// TwinCAT 3 PLC project Ampelschaltung
// libraries:
//   Tc2_Standard, * (Beckhoff Automation GmbH)
//   Tc2_Standard, * (Beckhoff Automation GmbH)
//   Tc2_System, * (Beckhoff Automation GmbH)
//   Tc2_System, * (Beckhoff Automation GmbH)
//   Tc3_Module, * (Beckhoff Automation GmbH)
//   Tc3_Module, * (Beckhoff Automation GmbH)
// project tree:
//   Global Variables/ Global_Variables.TcGVL, Variable_Configuration.TcGVL
//   / GlobalImagePool.TcGIPO (not stored), GlobalTextList.TcGTLO, Standard.TcTTO, Visualisierungsmanager.TcVMO (not stored)
//   POUs/ fb_Blink.TcPOU, MAIN.TcPOU
//   Visualizations/ Ende.TcVIS, Kreuzung.TcVIS

CONFIGURATION Ampelschaltung
    RESOURCE PLC ON TwinCAT3
        TASK Standard(INTERVAL := T#10ms, PRIORITY := 20);
        PROGRAM MAIN WITH Standard : MAIN;
    END_RESOURCE
END_CONFIGURATION

// ---- Global Variables/Global_Variables.TcGVL
{attribute 'Tc2GvlVarNames'}
VAR_GLOBAL
END_VAR

// ---- Global Variables/Variable_Configuration.TcGVL
{attribute 'Tc2GvlVarNames'}
VAR_CONFIG
END_VAR

// ---- POUs/MAIN.TcPOU
PROGRAM MAIN
VAR

	bON : BOOL;
	diStep : INT;
	bEndeInvisible : BOOL := TRUE;
	bOK : BOOL := FALSE;
	iPhase : REAL;
	bNacht : BOOL;

	(*Ampel Nord-Süd*)
	bNS_rot : BOOL;
	bNS_orange : BOOL;
	bNS_gruen : BOOL;

	(*Ampel West-Ost*)
	bWO_rot : BOOL;
	bWO_orange : BOOL;
	bWO_gruen : BOOL;

	(*Fussgängerampeln Nord-Süd*)
	bFGNS_rot : BOOL;
	bFGNS_gruen : BOOL;
	bFG : BOOL;

	(*Timer*)
	t1 : TON;

	t3 : TON;
	t2 : TON;

END_VAR

t1();

t3.IN := (t2.Q = FALSE);
t2.IN := t3.Q;

t3(PT:=T#3S);
t2(PT:=t#1s);


IF bON = TRUE AND diStep = 0
THEN
	diStep := 1000;

ELSIF bOn = FALSE
THEN
	diStep := 0;
END_IF


CASE diStep OF

0:
(*Idle*)
	bNS_rot:=FALSE;
	bNS_orange := FALSE;
	bNS_gruen := FALSE;

	bWO_rot:=FALSE;
	bWO_orange:=FALSE;
	bWO_gruen:=FALSE;
	bOK:=FALSE;
	bEndeInvisible := TRUE;

	bfgns_gruen := FALSE;
	bfgns_rot:= FALSE;

	t1.IN := FALSE;

	iPhase := 0;




1000:
(*Grünphase Nord-Süd, Rotphase West-Ost*)
	bNS_rot:=FALSE;
	bNS_orange := FALSE;
	bNS_gruen := TRUE;

	bWO_rot:=TRUE;
	bWO_orange:=FALSE;
	bWO_gruen:=FALSE;
	iPhase := 1;
	bfgns_rot := TRUE;

	t1.IN := TRUE;
	t1.PT := T#10000ms;

	IF bFG = TRUE
	THEN
		bfgns_gruen := TRUE;
		bfgns_rot:= FALSE;
	END_IF;

	IF bNacht = TRUE
	THEN
		diStep:=6000;
	END_IF

	IF t1.Q AND bnacht = TRUE
	THEN
		diStep := 6000;
	ELSIF t1.Q AND bNacht = FALSE
	THEN
		t1.IN := FALSE;
		bfgns_gruen := FALSE;
		bfgns_rot := TRUE;
		bFG := FALSE;
		diStep:= 2000;
	END_IF;


2000:
(*Orangephase Nord-Süd*)

	bNS_rot := FALSE;
	bNS_orange := TRUE;
	bNS_gruen := FALSE;

	bWo_rot :=TRUE;
	bWO_orange := TRUE;
	bWO_gruen :=FALSE;

	bFGNS_rot := TRUE;
	bFGNS_gruen := FALSE;

	iPhase := 2;

	t1(IN := bNS_orange, PT := T#5000ms);

		IF t1.Q
		THEN
			t1.IN := FALSE;
			diStep:= 3000;
	END_IF;


3000:
(*Rotphase Nord-Sued, Grünphase West-Ost*)

	bNS_rot:=TRUE;
	bNS_orange := FALSE;
	bNS_gruen := FALSE;

	bWO_rot:=FALSE;
	bWO_orange:=FALSE;
	bWO_gruen:=TRUE;
	iPhase := 3;
	bFGNS_rot := TRUE;

	t1(IN := bNS_rot, PT := T#5000ms);

	IF t1.Q
	THEN
		t1.IN := FALSE;
		diStep:= 4000;
	END_IF;

4000:
(*Rot-Orange-Phase Nord-Sued*)

	bNS_rot:=TRUE;
	bNS_orange := TRUE;
	bNS_gruen := FALSE;

	bWO_rot:=FALSE;
	bWO_orange:=TRUE;
	bWO_gruen:=FALSE;
	bFGNS_rot := TRUE;
	iPhase := 4;

	t1(IN := bNS_rot, PT := T#5000ms);

	IF t1.Q
	THEN
		t1.IN := FALSE;
		diStep:= 1000;
	END_IF;

6000:
(*Nachtmodus*)

	bNS_rot:=FALSE;
	bNS_orange := t3.Q;
	bNS_gruen := FALSE;
	
	bWO_rot:=FALSE;
	bWO_orange:= t3.Q;
	bWO_gruen:=FALSE;

	bFGNS_rot :=FALSE;
	bFGNS_gruen := FALSE;

	IF bNacht = FALSE
	THEN
		t1.IN := FALSE;
		diStep:= 1000;
	END_IF

(*5000:
(*Fenster Ende*)
	bEndeInvisible := FALSE;
	IF bOK
	THEN
		bEndeInvisible := TRUE;
		bON := FALSE;
		diStep := 0;
	END_IF;*)

END_CASE;

END_PROGRAM

// ---- POUs/fb_Blink.TcPOU
FUNCTION_BLOCK fb_Blink
VAR_INPUT
END_VAR
VAR_OUTPUT
END_VAR
VAR
		t1 : TON;
		t2 : TON;
END_VAR




t1.IN := (t2.Q = FALSE);

t2.IN := t1.Q;


t1(PT:=t#1s);
t2(PT:=t#2s); (*FEATUARE*) (*TEST*)

END_FUNCTION_BLOCK

// ---- GlobalTextList.TcGTLO
TEXTLIST GlobalTextList
  225 = 'Bitte drücken'
  117 = 'ENDE'
  226 = 'Nachtmodus'
  118 = 'OK'
  866 = 'ON'
END_TEXTLIST

// ---- Visualizations/Ende.TcVIS
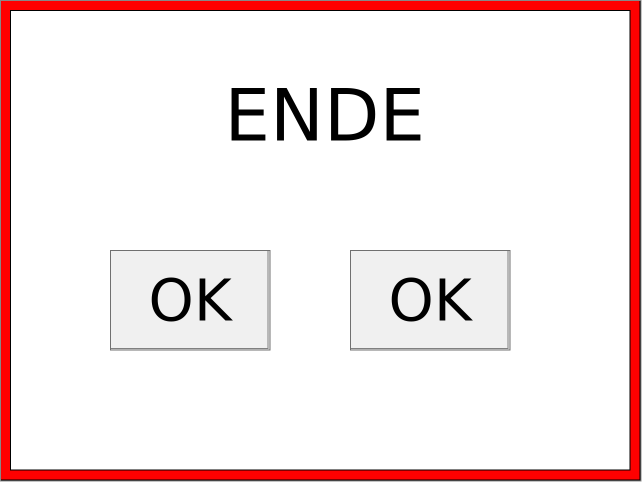
VISUALIZATION Ende  // 642x482
    Rectangle (0,0 640x480)
    Rectangle (10,10 620x460)
    Rectangle (130,50 390x130), "ENDE"
    Button (110,250 160x100), "OK"
        tap MAIN.bOK p1329445385=TRUE
    Button (350,250 160x100), "OK"
        tap MAIN.bOK p1329445385=TRUE
END_VISUALIZATION

// ---- Visualizations/Kreuzung.TcVIS
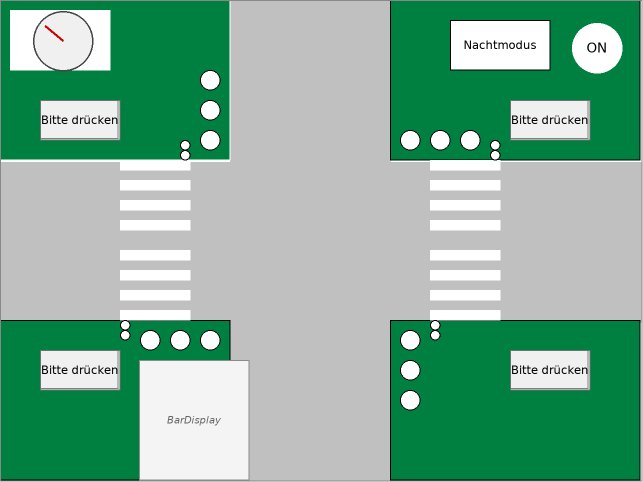
VISUALIZATION Kreuzung  // 643x482
    Rectangle (230,0 160x480)
    Rectangle (1,162 640x160)
    Rectangle (0,0 230x160)
    Rectangle (390,0 250x160)
        tap MAIN.bON
    Rectangle (390,320 250x160)
    Rectangle (0,320 230x160)
    Polyline (230,0)
    Polyline (630,160)
    Polyline (230,480)
    Polyline (630,320)
    Ellipse (200,330 20x20), colour toggle: MAIN.bWO_rot
    Ellipse (170,330 20x20), colour toggle: MAIN.bWO_orange
    Ellipse (140,330 20x20), colour toggle: MAIN.bWO_gruen
    Ellipse (400,360 20x20), colour toggle: MAIN.bNS_orange
    Ellipse (400,330 20x20), colour toggle: MAIN.bNS_rot
    Ellipse (460,130 20x20), colour toggle: MAIN.bWO_gruen
    Ellipse (430,130 20x20), colour toggle: MAIN.bWO_orange
    Ellipse (400,130 20x20), colour toggle: MAIN.bWO_rot
    Ellipse (400,390 20x20), colour toggle: MAIN.bNS_gruen
    Ellipse (200,130 20x20), colour toggle: MAIN.bNS_rot
    Ellipse (200,100 20x20), colour toggle: MAIN.bNS_orange
    Ellipse (200,70 20x20), colour toggle: MAIN.bNS_gruen
    Polyline (20,240)
    Polyline (60,240)
    Polyline (100,240)
    Polyline (140,240)
    Polyline (180,240)
    Polyline (220,240)
    Polyline (460,240)
    Polyline (540,240)
    Polyline (500,240)
    Polyline (580,240)
    Polyline (620,240)
    Polyline (310,340)
    Polyline (310,380)
    Polyline (310,420)
    Polyline (310,460)
    Polyline (310,480)
    Polyline (310,160)
    Polyline (310,120)
    Polyline (310,80)
    Polyline (310,40)
    Polyline (310,10)
    Ellipse (572,23 50x50), "ON", colour toggle: MAIN.bON
        toggle MAIN.bON
    Rectangle (10,10 100x60)
    Meter (13,11 100x60), value: MAIN.iPhase, scale format: %.1f, scale 0..4
    Rectangle (430,200 70x10)
    Rectangle (430,250 70x10)
    Rectangle (430,180 70x10)
    Rectangle (430,310 70x10)
    Rectangle (430,220 70x10)
    Rectangle (430,270 70x10)
    Rectangle (430,290 70x10)
    Rectangle (430,160 70x10)
    Polyline (420,240)
    Rectangle (120,200 70x10)
    Rectangle (120,250 70x10)
    Rectangle (120,180 70x10)
    Rectangle (120,310 70x10)
    Rectangle (120,220 70x10)
    Rectangle (120,270 70x10)
    Rectangle (120,290 70x10)
    Rectangle (120,160 70x10)
    Ellipse (120,330 10x10), colour toggle: MAIN.bFGNS_rot
    Ellipse (120,320 10x10), colour toggle: MAIN.bFGNS_gruen
    Ellipse (180,150 10x10), colour toggle: MAIN.bFGNS_gruen
    Ellipse (180,140 10x10), colour toggle: MAIN.bFGNS_rot
    Ellipse (430,330 10x10), colour toggle: MAIN.bFGNS_rot
    Ellipse (430,320 10x10), colour toggle: MAIN.bFGNS_gruen
    Ellipse (490,150 10x10), colour toggle: MAIN.bFGNS_gruen
    Ellipse (490,140 10x10), colour toggle: MAIN.bFGNS_rot
    Button (510,350 80x40), "Bitte drücken", pressed state: MAIN.bFG
        toggle MAIN.bFG
    Button (40,100 80x40), "Bitte drücken", pressed state: MAIN.bFG
        toggle MAIN.bFG
    Button (510,100 80x40), "Bitte drücken", pressed state: MAIN.bFG
        toggle MAIN.bFG
    Button (40,350 80x40), "Bitte drücken", pressed state: MAIN.bFG
        toggle MAIN.bFG
    RoundedRectangle (450,20 100x50), "Nachtmodus", colour toggle: MAIN.bNacht
        toggle MAIN.bNacht
    Rectangle (150,360 70x120)
    BarDisplay (139,360 110x120), value: MAIN.iPhase, scale format: %.1f, scale 0..4
END_VISUALIZATION
